// TwinCAT 3 PLC project HelloWorldPLC
// ProgramVersion: 3.1.4023.0
// libraries:
//   Tc2_Standard, * (Beckhoff Automation GmbH)
//   Tc2_System, * (Beckhoff Automation GmbH)
//   Tc3_Module, * (Beckhoff Automation GmbH)
//   Tc2_Utilities,3.3.52.0,Beckhoff Automation GmbH
//   Tc3_IotBase,3.1.19.0,Beckhoff Automation GmbH
// project tree:
//   DUTs/ Colors.TcDUT, complicatedFunc.TcPOU, funcWithReferences.TcPOU, MyStruct.TcDUT, sum.TcPOU
//   / PlcTask.TcTTO
//   POUs/ DataTypes.TcPOU, IDevice.TcIO, MAIN.TcPOU, Motor.TcPOU, ServoMotor.TcPOU, StructuresAndFunctions.TcPOU
// real-time tasks:
//   TASK PlcTask: cycle T#10ms, priority 20, ADS port 350

CONFIGURATION HelloWorldPLC
    RESOURCE PLC ON TwinCAT3
        TASK PlcTask(INTERVAL := T#10ms, PRIORITY := 20);
        PROGRAM MAIN WITH PlcTask : MAIN;
    END_RESOURCE
END_CONFIGURATION

// ---- DUTs/Colors.TcDUT
{attribute 'qualified_only'}
{attribute 'strict'}
TYPE Colors :
(
	Red,
	Green,
	Orange,
	Yellow
);
END_TYPE

// ---- DUTs/MyStruct.TcDUT
(* Some block comment for the struct *)
TYPE MyStruct :
STRUCT
	name : STRING;
	age : INT;
END_STRUCT
END_TYPE

// ---- POUs/IDevice.TcIO
INTERFACE IDevice

METHOD turnOn
VAR_INPUT
END_VAR
END_METHOD

END_INTERFACE

// ---- POUs/MAIN.TcPOU
PROGRAM MAIN
VAR
    someInt1 : INT := 20;
	someInt2 : INT := 10;
	result : INT;
	
	bigNum : INT;
	smallNum : INT;
	
	isCaluculated : BOOL := FALSE;
	isCompared : BOOL := FALSE;
	isIncreased : BOOL := FALSE;
	
	//timers
	//set timer for 3s
	fbTon : TON := (PT:=T#3S);
	trigger : BOOL := TRUE;
	isTimerDone : BOOL := FALSE;
END_VAR

IF NOT isCaluculated THEN
	result := sum(num1 := someInt1, num2 := someInt2);
	isCaluculated := TRUE;
END_IF

IF NOT isCompared THEN
	complicatedFunc(num1:=someInt1, num2:=someInt2, biggerNum=>bigNum, smallerNum=>smallNum);
	isCompared := TRUE;	
END_IF

IF NOT isIncreased THEN
	funcWithReferences(someInt1);
	isIncreased := TRUE;	
END_IF

//timers
//start timer when trigger is true
fbTon(IN:=trigger);
isTimerDone := fbTon.Q;

END_PROGRAM

// ---- DUTs/sum.TcPOU
FUNCTION sum : INT
VAR_INPUT
	num1 : INT;
	num2 : INT;
END_VAR
VAR
END_VAR

sum := num1 + num2;

END_FUNCTION

// ---- DUTs/complicatedFunc.TcPOU
FUNCTION complicatedFunc : INT
VAR_INPUT
	num1 : INT;
	num2 : INT;
END_VAR
VAR
END_VAR
VAR_OUTPUT
	biggerNum : INT;
	smallerNum : INT;
END_VAR

IF num1 > num2 THEN
	biggerNum := num1;
	smallerNum := num2;
ELSE
	biggerNum := num2;
	smallerNum := num1;
END_IF

END_FUNCTION

// ---- DUTs/funcWithReferences.TcPOU
FUNCTION funcWithReferences : INT
VAR_IN_OUT
	num : INT;
END_VAR
VAR
END_VAR

num := num+1;

END_FUNCTION

// ---- POUs/DataTypes.TcPOU
PROGRAM DataTypes
VAR
	floatExample : REAL;
	someStr : STRING;
	someInt : INT := 20;
	{REFERENCE TO someInt}
	refInt : REFERENCE TO INT REF=someInt;
	
	bytesCountFloat : UINT;
	bytesCountInt : UINT;
	bytesCountStr : UINT;
	
	{U may declare negative indexes : [-5..4]}
	someArr : ARRAY[1..5] OF INT := [10, 20, 30, 40, 50];
	twoDemArr : ARRAY [0..3, 0..9] OF REAL;
END_VAR

bytesCountFloat := SIZEOF(floatExample);
bytesCountStr := SIZEOF(someStr);
bytesCountInt := SIZEOF(someInt);

someArr[2] := 0;

END_PROGRAM

// ---- POUs/Motor.TcPOU
FUNCTION_BLOCK Motor IMPLEMENTS IDevice
VAR_INPUT
END_VAR
VAR_OUTPUT
END_VAR
VAR
	isOn : BOOL := FALSE;       
END_VAR

METHOD PUBLIC turnOn
VAR_INPUT
END_VAR
isOn := true;
END_METHOD

END_FUNCTION_BLOCK

// ---- POUs/ServoMotor.TcPOU
FUNCTION_BLOCK ServoMotor EXTENDS Motor
VAR_INPUT
END_VAR
VAR_OUTPUT
END_VAR
VAR
	position : INT;
END_VAR

METHOD turn90Deg
VAR_INPUT
END_VAR
position := 90;
END_METHOD

END_FUNCTION_BLOCK

// ---- POUs/StructuresAndFunctions.TcPOU
PROGRAM StructuresAndFunctions
VAR
	myStruct : MyStruct;
	
	age : INT;
	name : STRING;
END_VAR

age := myStruct.age;
name := myStruct.name;

END_PROGRAM
